// TIA Portal V20 export
// export: Created 2026-07-14T13:44:08.6532919Z, ExportSetting WithDefaults, DisplayName Totally Integrated Automation Portal, DisplayVersion V20 Update 5, DisplayName TIA Portal Openness, DisplayVersion V20 Update 4, DisplayName TIA Portal Version Control Interface, DisplayVersion V20 Update 5, DisplayName SINAMICS Startdrive Advanced, DisplayVersion V20, DisplayName SINAMICS DCC, DisplayVersion V20, DisplayName SINAMICS Startdrive G130, G150, S120, S150, SINAMICS MV, G220, S200, S210, DisplayVersion V20, DisplayName SINAMICS Startdrive G110M, G120, G120C, G120D, G120P, G115D, DisplayVersion V20, DisplayName STEP 7 Professional, DisplayVersion V20 Update 5, DisplayName STEP 7 Safety, DisplayVersion V20 Update 2, DisplayName WinCC Basic/Comfort/Advanced, DisplayVersion V20 Update 5, DisplayName WinCC Unified, DisplayVersion V20 Update 5
FUNCTION "ThresholdAlarms" : Void   // FC20, LAD
{ S7_Optimized_Access := 'TRUE' }
VERSION : 0.1
// Threshold/comparison reference examples (Eq/Ge/Lt/Ne/Gt/Le)
// stored: AutoNumber true, IsIECCheckEnabled false, SetENOAutomatically false, UDAEnableTagReadback false
   VAR_TEMP
      ModeSelect : Int;
      AutoModeEnable : Bool;
      AutoModeActive : Bool;
      TankLevelHighEnable : Bool;
      TankLevel : Int;
      TankLevelHighAlarm : Bool;
      TankLevelLowEnable : Bool;
      TankLevelLowAlarm : Bool;
      FaultCheckEnable : Bool;
      StatusWord : Int;
      FaultPresent : Bool;
      PressureHighEnable : Bool;
      Pressure : Int;
      PressureHighAlarm : Bool;
      PressureLowEnable : Bool;
      PressureLowAlarm : Bool;
   END_VAR
BEGIN

REGION Network 1: Mode selection (Eq)
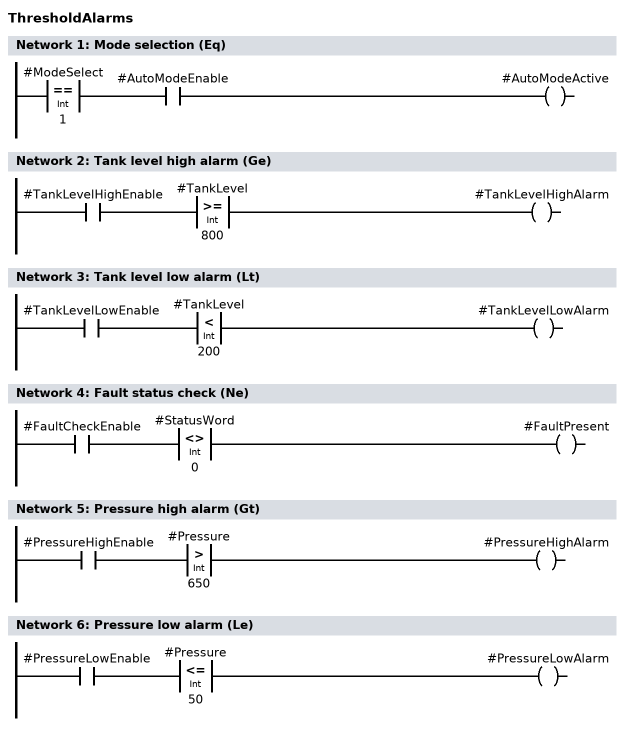
   RUNG wire#powerrail
      { S7_Templates := "SrcType := Int" } EQ_Contact(in1 := #ModeSelect, in2 := 1)
      Contact( #AutoModeEnable )
      Coil( #AutoModeActive )
   END_RUNG
   // the same network as SCL:
   #AutoModeActive := (#ModeSelect = 1) AND #AutoModeEnable;
END_REGION

REGION Network 2: Tank level high alarm (Ge)
   RUNG wire#powerrail
      Contact( #TankLevelHighEnable )
      { S7_Templates := "SrcType := Int" } GE_Contact(in1 := #TankLevel, in2 := 800)
      Coil( #TankLevelHighAlarm )
   END_RUNG
   // the same network as SCL:
   #TankLevelHighAlarm := #TankLevelHighEnable AND (#TankLevel >= 800);
END_REGION

REGION Network 3: Tank level low alarm (Lt)
   RUNG wire#powerrail
      Contact( #TankLevelLowEnable )
      { S7_Templates := "SrcType := Int" } LT_Contact(in1 := #TankLevel, in2 := 200)
      Coil( #TankLevelLowAlarm )
   END_RUNG
   // the same network as SCL:
   #TankLevelLowAlarm := #TankLevelLowEnable AND (#TankLevel < 200);
END_REGION

REGION Network 4: Fault status check (Ne)
   RUNG wire#powerrail
      Contact( #FaultCheckEnable )
      { S7_Templates := "SrcType := Int" } NE_Contact(in1 := #StatusWord, in2 := 0)
      Coil( #FaultPresent )
   END_RUNG
   // the same network as SCL:
   #FaultPresent := #FaultCheckEnable AND (#StatusWord <> 0);
END_REGION

REGION Network 5: Pressure high alarm (Gt)
   RUNG wire#powerrail
      Contact( #PressureHighEnable )
      { S7_Templates := "SrcType := Int" } GT_Contact(in1 := #Pressure, in2 := 650)
      Coil( #PressureHighAlarm )
   END_RUNG
   // the same network as SCL:
   #PressureHighAlarm := #PressureHighEnable AND (#Pressure > 650);
END_REGION

REGION Network 6: Pressure low alarm (Le)
   RUNG wire#powerrail
      Contact( #PressureLowEnable )
      { S7_Templates := "SrcType := Int" } LE_Contact(in1 := #Pressure, in2 := 50)
      Coil( #PressureLowAlarm )
   END_RUNG
   // the same network as SCL:
   #PressureLowAlarm := #PressureLowEnable AND (#Pressure <= 50);
END_REGION
END_FUNCTION
